Staubli VAL3: getRobotArea.pgx

public program getRobotArea(num x_nConvNum (dimensions=1), num& x_nAreaNumber[] (dimensions=1))
begin
  // This program returns in which area number is currently located
  //
  // Input Param
  // x_nConvNum    : Conveyor number
  //
  // Output param
  // x_nAreNumber  : Number of the area in hich is the robot
  //           --> -1: Invalid parameter
  //           --> 0 : robot is beside or above the conveyor
  //           --> 1 : Robot is upstream of the upstream end of the tracking window
  //           --> 2 : Robot is within tracking window
  //           --> 3 : Robot is downstream of the downstream end of the tracking window
  //
  //----------------------------------------------------------------
  //
  if (x_nConvNum>0) and (x_nConvNum<=size(nTrackingZone)-1)
    x_nAreaNumber=nTrackingZone[x_nConvNum]
  else
    x_nAreaNumber=-1
  endIf
end
